{attribute 'linkalways'} 
{attribute 'no_explicit_call' := 'This FB is a CLASS and must be accessed using methods or properties'}
{attribute 'enable_dynamic_creation'}
FUNCTION_BLOCK _ETcVnEdgeDirection EXTENDS EnumDatatypeBase
VAR
	localData : ETcVnEdgeDirection;
	activeData : REFERENCE TO ETcVnEdgeDirection;
	enumBaseDatatype : _DINT(localData);
END_VAR

METHOD PRIVATE AddLocalEnumeration
VAR_INPUT
	Enumeration : T_MAXSTRING;
	Value : ETcVnEdgeDirection;
END_VAR
AddEnumeration(Enumeration, Value);
END_METHOD

PROPERTY PUBLIC Address : PVOID
GET
Address := ADR(activeData);
END_GET
END_PROPERTY

METHOD PUBLIC ClearReference
VAR_INPUT
END_VAR
activeData REF= localData;
SetBaseDatatypeReference();
END_METHOD

METHOD PUBLIC Clone : I_Datatype
VAR
    pClone : POINTER TO _ETcVnEdgeDirection;
END_VAR
pClone := __NEW(_ETcVnEdgeDirection(InitialValue := Value));
Clone := pClone^;
END_METHOD

METHOD FB_init : BOOL
VAR_INPUT
	bInitRetains : BOOL; // if TRUE, the retain variables are initialized (warm start / cold start)
	bInCopyCode : BOOL;  // if TRUE, the instance afterwards gets moved into the copy code (online change)
	InitialValue : ETcVnEdgeDirection;
END_VAR
localData := InitialValue;
AddBaseDatatype(enumBaseDatatype);
ClearReference();

AddLocalEnumeration('TCVN_ED_DARK_TO_LIGHT', ETcVnEdgeDirection.TCVN_ED_DARK_TO_LIGHT);
AddLocalEnumeration('TCVN_ED_LIGHT_TO_DARK', ETcVnEdgeDirection.TCVN_ED_LIGHT_TO_DARK);
END_METHOD

PROPERTY PUBLIC Identifier : T_MAXSTRING
GET
Identifier := 'ETcVnEdgeDirection';
END_GET
END_PROPERTY

METHOD IsEnumeratorValueEqual : BOOL
VAR_INPUT
	Enumerator : I_KeyValueForwardEnumerator;
END_VAR
VAR
	storedValue : ETcVnEdgeDirection;
END_VAR
IF NOT Enumerator.TryGet(storedValue) THEN
	RETURN;
END_IF

IsEnumeratorValueEqual := storedValue = activeData;
END_METHOD

METHOD PUBLIC MakeReferenceTo
VAR_INPUT
	ReferenceTarget : REFERENCE TO ETcVnEdgeDirection;
END_VAR
activeData REF= ReferenceTarget;
SetBaseDatatypeReference();
END_METHOD

METHOD PROTECTED SetBaseDatatypeReference
VAR_INPUT
END_VAR
enumBaseDatatype.MakeReferenceTo(activeData);
END_METHOD

PROPERTY PUBLIC Size : UDINT
GET
Size := SIZEOF(activeData);
END_GET
END_PROPERTY

METHOD TryMakeReferenceTo : BOOL
VAR_INPUT
	Target : I_Datatype;
END_VAR
VAR
	pTargetData : POINTER TO ETcVnEdgeDirection;
END_VAR
IF NOT IsEquivalentTo(Target) THEN
	RETURN;
END_IF

pTargetData := Target.Address;
activeData REF= pTargetData^;
SetBaseDatatypeReference();
TryMakeReferenceTo := TRUE;
END_METHOD

PROPERTY PUBLIC Value : ETcVnEdgeDirection
GET
Value := activeData;
END_GET
SET
activeData := Value;
END_SET
END_PROPERTY

END_FUNCTION_BLOCK

(* stored: Version 1.1.0.1, ProductVersion 3.1.4024.13
   POU _ETcVnEdgeDirection: Id {34f9a536-f1f5-0489-11b4-43cfbbe26369}, SpecialFunc None
   Folder Core: Id {58e12531-754a-0666-3b44-bce0a75308ba}
   Folder Protected: Id {f8b79d82-ae18-0f54-2e80-e4ea0db2c8a5}
   Folder Customize: Id {7d1db118-e145-06d0-2af9-ee2b91d40590}
   Folder Constructor: Id {ab78af80-ede1-07cc-3544-57ebe611c29e}
   Folder Private: Id {3bf217fc-19e8-0c41-32e8-fa11b1479b34}
   Folder Protected: Id {dae23890-d50d-009f-2136-4b5a5c743612}
   Method AddLocalEnumeration: Id {f47c54ee-ea3c-01fd-3a5d-0c7056ae0bf3}
   Property Address: Id {a6b2e1a1-8290-0c9a-367e-79f45ccdbac2}
   Get Get: Id {f10baab7-a921-0126-0307-0765c360df9a}
   Method ClearReference: Id {9da33047-8402-04e5-39a0-b832c7bfdd1a}
   Method Clone: Id {e66af5ce-18a6-04d3-1511-0d7d052b3abb}
   Method FB_init: Id {1cb4c907-b356-09d9-2a9e-2d472bd95fee}
   Property Identifier: Id {e8b8bc8b-531e-0591-11ab-f0b7b87e0e5f}
   Get Get: Id {44d06f23-b5e7-0664-1fa1-b386a49fb736}
   Method IsEnumeratorValueEqual: Id {54a754fb-e093-0741-21c3-9e525c70c4a4}
   Method MakeReferenceTo: Id {3fd45972-d583-0067-3728-c73e981a03fe}
   Method SetBaseDatatypeReference: Id {ee374003-e442-017b-3735-853a9e4316de}
   Property Size: Id {1ed940a8-41f8-0156-10f2-466713e75f5c}
   Get Get: Id {08b915a5-5d85-05b3-17ce-0c98f3632f60}
   Method TryMakeReferenceTo: Id {7c71209a-c62a-0685-107c-c2b2a43e72d0}
   Property Value: Id {05ef739d-89fb-01b2-0540-cae8ecd16b58}
   Get Get: Id {014b8e07-f525-00af-3629-3f433b61faf8}
   Set Set: Id {5b8a49ee-b548-028d-0cbe-b9b64e96471c} *)
